Universal Robots URScript: go_to_home.urscript

def go_to_home():
	movel(p[-0.171, -0.682, 0.428, 0, 3.14, 0], a=1.0, v=0.8)
end
